PROGRAM B_3_1_PRG_Master_Station_3

VAR
	eState								: E_Station2_State;
	tonErrorReset						: TON;
	tonStationStopped					: TON;
	ctuErrorCounter						: CTU;
	rGoodStatistics						: R_TRIG;
	rBadStatistics						: R_TRIG;
	rEfficency							: STRING(510);
	
	bPersistentError					: bool;
/////////////////////////////////////////////////////////////////////////////////////I O/////////////////////////////////////////////////////////////////////////////////////	
	bStopped							: BOOL;
	bError								: BOOL;
	bReady								: BOOL;
	bDone								: BOOL;
	bPass								: BOOL;
	bFail								: BOOL;
	
END_VAR

VAR_INPUT	
	
	CMD									:ST_StationCMD;	
	
END_VAR

VAR_OUTPUT	
	
	STATUS								:ST_StationStatus;	
	
END_VAR

B_3_2_PRG_Fault_Station_3( aAlarms := stAlarms );
a_ACT_Ctrl_Station_3();
b_ACT_IO();
c_ACT_Statistics_Station_3();

ACTION a_ACT_Ctrl_Station_3:
/////////////////////////////////////////////////////////////////////////////////////UTILITIES/////////////////////////////////////////////////////////////////////////////////////
tonErrorReset( IN := (eState = E_Station3_State.RESET_ERROR), PT := T#500MS);
tonStationStopped( IN := bStopped, PT := T#1S);
ctuErrorCounter( CU := eState = E_Station3_State.RESET_ERROR, RESET := ((ctuErrorCounter.CV = 5) AND eState = E_Station3_State.PERSISTENT_ERROR), PV := 5, Q => bPersistentError);

/////////////////////////////////////////////////////////////////////////////////////CONDITIONS/////////////////////////////////////////////////////////////////////////////////////

IF (CMD.bAbort OR bError) AND ( eState			= E_Station3_State.HOMING OR
								eState			= E_Station3_State.READY OR
								eState			= E_Station3_State.MOVEMENT_A OR
								eState			= E_Station3_State.MOVEMENT_B OR
								eState			= E_Station3_State.MOVEMENT_C OR
								eState			= E_Station3_State.READY OR
								eState			= E_Station3_State.DONE) THEN
								
	eState						:= E_Station3_State.STOPPING;
	
END_IF

IF CMD.bAbort OR NOT CMD.bEnable THEN
	eState						:= E_Station3_State.ABORTED;
END_IF

CASE eState OF
	
	E_Station3_State.ABORTED:
								IF CMD.bEnable AND NOT bError THEN
									eState						:= E_Station3_State.HOMING;
								ELSIF bError THEN
									eState						:= E_Station3_State.ERROR;
								END_IF
	
	E_Station3_State.HOMING:
								IF bReady THEN
									eState						:= E_Station3_State.READY;
								END_IF
	E_Station1_State.RESET:
								stCycleDataStation3.bPass	:= FALSE;
								stCycleDataStation3.bFail	:= FALSE;
								
								eState						:= E_Station3_State.READY;	
	E_Station3_State.READY:
								IF CMD.bExecute AND stStation3.Mov1 THEN
									eState						:= E_Station3_State.MOVEMENT_A;
								ELSIF CMD.bExecute AND stStation3.Mov2 THEN
									eState						:= E_Station3_State.MOVEMENT_B;
								ELSIF CMD.bExecute AND stStation3.Mov3 THEN
									eState						:= E_Station3_State.MOVEMENT_C;
								END_IF
	
	E_Station3_State.MOVEMENT_A:
								IF bDone AND stStation3.Mov1 THEN
									eState						:= E_Station3_State.DONE;
								END_IF
	
	E_Station3_State.MOVEMENT_B:
								IF bDone AND stStation3.Mov2 THEN
									eState						:= E_Station3_State.DONE;
								END_IF
	E_Station3_State.MOVEMENT_C:
								IF bDone AND stStation3.Mov3 THEN
									eState						:= E_Station3_State.DONE;
								END_IF
	E_Station3_State.DONE:
								IF  CMD.bReady THEN
									eState						:= E_Station3_State.READY;
								END_IF
								
	E_Station1_State.RESULTS:
								
								IF bPass THEN
									stCycleDataStation3.bPass	:= TRUE;
								ELSIF bFail THEN
								 	stCycleDataStation3.bFail	:= TRUE;
								END_IF
								
								IF  CMD.bEndCycle THEN
									eState						:= E_Station3_State.RESET;
								END_IF
	/////////////////////////////////////////////////////////////////////////////////////RESET CMD/////////////////////////////////////////////////////////////////////////////////////
	
	E_Station3_State.STOPPING: 
								IF tonStationStopped.Q THEN
									IF bError THEN
										eState						:= E_Station3_State.ERROR;
									ELSE eState						:= E_Station3_State.ABORTED;
									END_IF

								END_IF
	
	E_Station3_State.ERROR:
								IF NOT bError THEN
									eState						:= E_Station3_State.ABORTED;
								ELSE eState						:= E_Station3_State.RESET_ERROR;
								END_IF
	
	E_Station3_State.RESET_ERROR:
								IF tonErrorReset.Q AND NOT bPersistentError THEN
									eState						:= E_Station3_State.ERROR;
								ELSIF bPersistentError THEN
									eState						:= E_Station3_State.PERSISTENT_ERROR;
								END_IF
	
	E_Station3_State.PERSISTENT_ERROR:
								IF CMD.bReset THEN
									eState						:= E_Station3_State.ERROR;
								END_IF
								
								

ELSE eState := E_Station3_State.ABORTED;
	
END_CASE
/////////////////////////////////////////////////////////////////////////////////////STATUS/////////////////////////////////////////////////////////////////////////////////////

Status.bBusy				:= 	eState			= E_Station3_State.HOMING OR
								eState			= E_Station3_State.MOVEMENT_A OR
								eState			= E_Station3_State.MOVEMENT_B OR
								eState			= E_Station3_State.MOVEMENT_C OR
								eState			= E_Station3_State.STOPPING;
								
Status.bDone				:=	eState			= E_Station3_State.DONE;
											
Status.bError				:= 	eState			= (E_Station3_State.ERROR OR  E_Station3_State.RESET_ERROR OR E_Station3_State.PERSISTENT_ERROR);

Status.bReady				:= 	eState			= E_Station3_State.READY;

Status.bStopped				:= 	eState			= E_Station3_State.ABORTED OR
								eState			= E_Station3_State.READY OR
								eState			= E_Station3_State.ERROR OR
								eState			= E_Station3_State.RESET_ERROR;
END_ACTION

ACTION b_ACT_IO:
//bStopped								:=;
//bError								:=;
//bReady								:=;
//bDone
END_ACTION

ACTION c_ACT_Statistics_Station_3:
stStatisticsHMI[3].sName			:= 'Station 3';


rGoodStatistics( CLK := (stCycleDataStation3.bPass AND (eState = E_Station3_State.RESULTS)) OR bStatisticsTest[4]);
rBadStatistics( CLK := (stCycleDataStation3.bFail AND (eState = E_Station3_State.RESULTS)) OR bStatisticsTest[5]);

IF 	rGoodStatistics.Q THEN
	
	stStatisticsHMI[3].nGood		:= stStatisticsHMI[3].nGood + 1;
	stStatisticsHMI[3].nTotalGood	:= stStatisticsHMI[3].nTotalGood + 1;
	
END_IF
								
IF 	rBadStatistics.Q THEN
	
	stStatisticsHMI[3].nBad			:= stStatisticsHMI[3].nBad + 1;
	stStatisticsHMI[3].nTotalBad	:= stStatisticsHMI[3].nTotalBad + 1;
	
END_IF

IF stStatisticsHMI[3].bResetGood THEN
	stStatisticsHMI[3].nGood		:= 0;
END_IF

IF stStatisticsHMI[3].bResetBad THEN
	stStatisticsHMI[3].nBad			:= 0;
END_IF

IF (( stStatisticsHMI[3].nGood + stStatisticsHMI[3].nBad) <> 0) THEN
	
	rEfficency							:= LREAL_TO_FMTSTR(in := (DINT_TO_REAL(stStatisticsHMI[3].nGood) /( DINT_TO_REAL(stStatisticsHMI[3].nGood) + DINT_TO_REAL(stStatisticsHMI[3].nBad))) * 100.0,iPrecision := 2, bRound := TRUE);
	stStatisticsHMI[3].nEfficency		:= CONCAT(STR1 := '%', STR2 := (rEfficency));

ELSE stStatisticsHMI[3].nEfficency		:= CONCAT(STR1 := '%', STR2 := (DINT_TO_STRING(0)));
	
END_IF
END_ACTION

END_PROGRAM

(* stored: Version 1.1.0.1, ProductVersion 3.1.4024.13
   POU B_3_1_PRG_Master_Station_3: Id {474f4225-5110-4ccd-bbcf-78541da80fa5}, SpecialFunc None
   Action a_ACT_Ctrl_Station_3: Id {18b6a780-51d7-4962-ac1f-d8e3484c4d5a}
   Action b_ACT_IO: Id {440050ef-4990-4273-9ec8-027f575cfd9b}
   Action c_ACT_Statistics_Station_3: Id {b9943b98-9d8e-469d-a7a3-a69e1222f6e9} *)
